# EPICS StreamDevice protocol: scu800App/Db/edwards.proto
Terminator   = "";
#LockTimeout  = 500;
ReplyTimeout = 200;
ReadTimeout  = 200;
WriteTimeout = 100;
MaxInput     = 180;
#ExtraInput   = Error;
ExtraInput   = Ignore;

wCtrl {
  out ${1} 2 "%.2r";
}

rCtrl {
  out ${1} 2;
  in  "%02r";
}

rConv {
  out ${1} 0;
  in  "%02r";
}
## e.g Command("01") {
Command {
    out "@\$1",STX,"001 E%02X",ETX,"%3<xor8ff>";
    in ACK,$1,STX,"001#",ETX,"%6<xor8ff>";
    out ACK,$1;
}
ReadMotorTemp {
    MaxInput = 18;
    ExtraInput  = Error;
    out        "@",$1,STX,"001?e",ETX,"%3<xor8ff>";
    in  ACK,$1,"@",$1,STX,"001 e%!4X",ETX,"%6<xor8ff>";
    out ACK,$1;
}
#ReadSetpoint: No reply within 200 ms to "@<01><02>001?d<03><96>"
#StreamIoTimeout input="01@01<02>001 d012C003C<03><8b>", size=21)
ReadSetPoint {
    MaxInput = 22;
    out "@",$1,STX,"001?d",ETX,"%3<xor8ff>";
    in ACK,$1,"@",$1,STX,"001 d%4X%*4X",ETX,"%6<xor8ff>";
    out ACK,$1;
}
ReadSetPointTMS {
    MaxInput = 22;
    in ACK,$1,"@",$1,STX,"001 d%*4X%4X",ETX,"%6<xor8ff>";
}
#out "@",$1,STX,"001?h",ETX,"%3<xor8ff>";
ReadSpeedSetPoint{
    MaxInput = 18;
    out "@",$1,STX,"001?h",ETX,"%3<xor8ff>";
    in  ACK,$1,"@",$1,STX,"001 h%!4X",ETX,"%6<xor8ff>";
    out ACK,$1;
}
# e.g SetSpeedSetPoint("01") {
#NOK    @init {ReadSpeedSetPoint($1); }
SetSpeedSetPoint {
    MaxInput = 13;
    out "@",$1,STX,"001 h%04X",ETX,"%3<xor8ff>";
    in ACK,$1,"@",$1,STX,"001#",ETX,"%6<xor8ff>";
    out ACK,$1;
}
ReadStatus {
    MaxInput = 22;
#    ReplyTimeout = 300;
    out        "@",$1,STX,"001?f",ETX,"%3<xor8ff>";
    in  ACK,$1,"@",$1,STX,"001 f%!8X",ETX,"%6<xor8ff>";
    out ACK,$1;
}
ReadStatusRMode {
#    ReplyTimeout = 300;
    MaxInput = 22;
    in  ACK,$1,"@",$1,STX,"001 f%!2X%*6X",ETX,"%6<xor8ff>";
}
ReadStatusTMSEnable {
    MaxInput = 22;
    in  ACK,$1,"@",$1,STX,"001 f%%*2X!2X%*4X",ETX,"%6<xor8ff>";
}
ReadStatusINHIBITEnable {
    MaxInput = 22;
    in  ACK,$1,"@",$1,STX,"001 f%%*4X!2X%*2X",ETX,"%6<xor8ff>";
}

ReadMeas {
    out "@",$1,STX,"001?D",ETX,"%3<xor8ff>";
    in  ACK,$1,"@",$1,STX,"001 D%*14X%!4X",ETX,"%6<xor8ff>";
    out ACK,$1;
}
ReadModFonct {
    MaxInput = 172;
    out        "@",$1,STX,"001?M",ETX,"%3<xor8ff>";
    in  ACK,$1,"@",$1,STX,"001 M%!2X%*156X",ETX,"%6<xor8ff>";
    out ACK,$1;
}
ReadModFonctNErrors {
#    ExtraInput = Ignore;
    MaxInput = 172;
    in  ACK,$1,"@",$1,STX,"001 M%*!2X%!2X%*154X",ETX,"%6<xor8ff>";
}
ReadModFonctError1 {
#    ExtraInput = Ignore;
    MaxInput = 172;
    in  ACK,$1,"@",$1,STX,"001 M%*!4X%!2X%*152X",ETX,"%6<xor8ff>";
}
ReadModFonctError2 {
    MaxInput = 172;
    in  ACK,$1,"@",$1,STX,"001 M%*!6X%!2X%*150X",ETX,"%6<xor8ff>";
}
## OK
ReadModFonctWWarning {
    ExtraInput = Ignore;
    MaxInput = 176;
    out        "@",$1,STX,"001?m",ETX,"%3<xor8ff>";
    in  ACK,$1,"@",$1,STX,"001 m%!2X%*160c",ETX,"%6<xor8ff>";
    out ACK,$1;
}
# NOK
ReadWarning {
    ExtraInput = Ignore;
    MaxInput = 176;
    in  ACK,$1,"@",$1,STX,"001 m%*!2X%!4X%*156c",ETX,"%6<xor8ff>";
}
ReadModFonctWWarningNErrors {
    MaxInput = 176;
    in  ACK,$1,"@",$1,STX,"001 m%*!6X%!2X%*154c",ETX,"%6<xor8ff>";
}
# Connect a stringout record to this to get
# a generic command interface.
# After processing finishes, the record contains the reply.

debug {
    ExtraInput = Ignore;
    out "%s"; in "%60c"
}
